// TwinCAT 3 PLC project Untitled1
// ProgramVersion: 3.1.4024.0
// libraries:
//   Tc2_Standard, * (Beckhoff Automation GmbH)
//   Tc2_System, * (Beckhoff Automation GmbH)
//   Tc3_Module, * (Beckhoff Automation GmbH)
// project tree:
//   / GlobalTextList.TcGTLO (not stored), PlcTask.TcTTO (not stored), Visualization Manager.TcVMO (not stored)
//   GVLs/ GIOL.TcGVL (not stored), Global_IO_assignment.TcPOU (not stored), GVL.TcGVL (not stored)
//   POUs/ MAIN.TcPOU, INMODE.TcPOU (not stored)
//   VISUs/ StandardPLCversenyVISU.TcVIS
// real-time tasks:
//   TASK PlcTask: cycle T#10ms, priority 20, ADS port 350
// I/O:
//   DEVICE Device 1 (EtherCAT), AmsNetId 5.86.98.224.2.1
//     Term 1 (EK1200) [EK1200-5000 EtherCAT Power supply (2A E-Bus)]
//       Term 2 (EL1008) [EL1008 8Ch. Dig. Input 24V, 3ms]
//       Term 3 (EL1008) [EL1008 8Ch. Dig. Input 24V, 3ms]
//       Term 4 (EL2008) [EL2008 8Ch. Dig. Output 24V, 0.5A]
//       Term 5 (EL2008) [EL2008 8Ch. Dig. Output 24V, 0.5A]
//       Term 6 (EL9011) [EL9011 End Terminal]
// variable links:
//   Untitled1/Untitled1 Instance <-> Device 1 (EtherCAT)/Term 1 (EK1200)/Term 2 (EL1008)
//     PlcTask Inputs/GIOL.xIn{0..7} <-> Channel {1..8}/Input  (8 links)
//   Untitled1/Untitled1 Instance <-> Device 1 (EtherCAT)/Term 1 (EK1200)/Term 3 (EL1008)
//     PlcTask Inputs/GIOL.xIn{8..15} <-> Channel {1..8}/Input  (8 links)
//   Untitled1/Untitled1 Instance <-> Device 1 (EtherCAT)/Term 1 (EK1200)/Term 4 (EL2008)
//     PlcTask Outputs/GIOL.Out{0..7} <-> Channel {1..8}/Output  (8 links)
//   Untitled1/Untitled1 Instance <-> Device 1 (EtherCAT)/Term 1 (EK1200)/Term 5 (EL2008)
//     PlcTask Outputs/GIOL.Out{8..15} <-> Channel {1..8}/Output  (8 links)

// ---- POUs/MAIN.TcPOU
PROGRAM MAIN
VAR
	INMODE : INMODE;
END_VAR

INMODE(); 
CASE GIOL.CaseNum OF
	0:GIOL.TaskName:="First Tsak";
	10:GIOL.TaskName:="Second Tsak";
	20:GIOL.TaskName:="Third Tsak";
	30:GIOL.TaskName:="Fourth Tsak";
	40:GIOL.TaskName:="Fifth Tsak";
	50:GIOL.TaskName:="Sixth Tsak";
	ELSE
		GIOL.CaseNum:=0;
END_CASE

END_PROGRAM

// ---- VISUs/StandardPLCversenyVISU.TcVIS
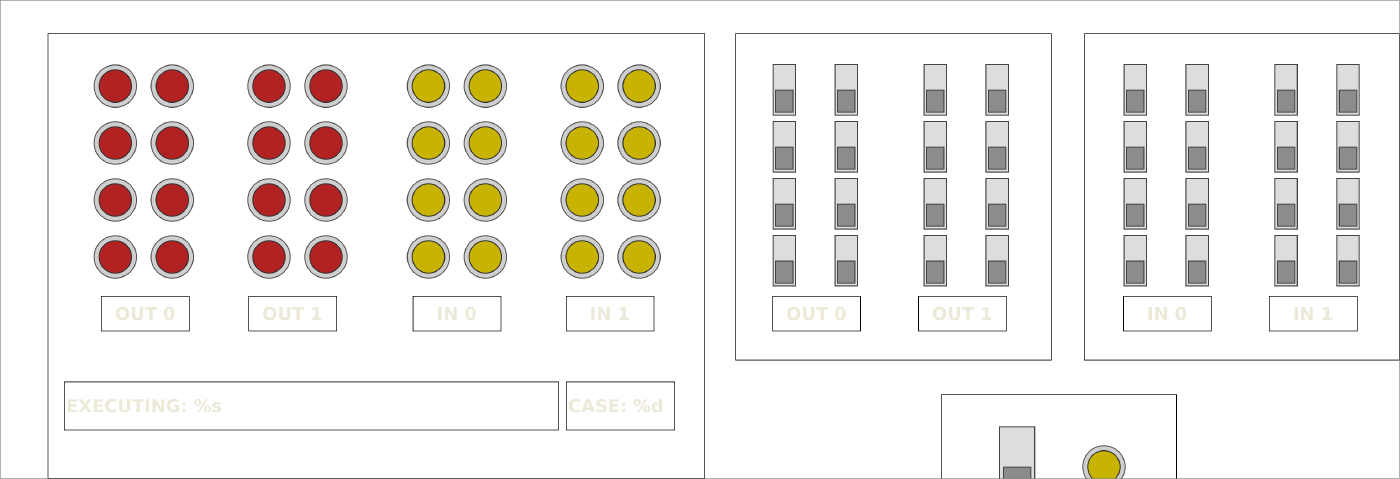
VISUALIZATION StandardPLCversenyVISU  // 1967x673
    Rectangle (1322,554 331x259)
    Rectangle (1033,47 444x459)
    Rectangle (67,47 923x626)
    Lamp1 (127,86 70x70), variable: GIOL.out0, style: Lamp-Lamp1-Red
    Lamp1 (207,86 70x70), variable: GIOL.out1, style: Lamp-Lamp1-Red
    Lamp1 (343,86 70x70), variable: GIOL.out8, style: Lamp-Lamp1-Red
    Lamp1 (423,86 70x70), variable: GIOL.out9, style: Lamp-Lamp1-Red
    Lamp1 (127,166 70x70), variable: GIOL.out2, style: Lamp-Lamp1-Red
    Lamp1 (207,166 70x70), variable: GIOL.out3, style: Lamp-Lamp1-Red
    Lamp1 (343,166 70x70), variable: GIOL.out10, style: Lamp-Lamp1-Red
    Lamp1 (423,166 70x70), variable: GIOL.out11, style: Lamp-Lamp1-Red
    Lamp1 (127,246 70x70), variable: GIOL.out4, style: Lamp-Lamp1-Red
    Lamp1 (207,246 70x70), variable: GIOL.out5, style: Lamp-Lamp1-Red
    Lamp1 (343,246 70x70), variable: GIOL.out12, style: Lamp-Lamp1-Red
    Lamp1 (423,246 70x70), variable: GIOL.out13, style: Lamp-Lamp1-Red
    Lamp1 (127,326 70x70), variable: GIOL.out6, style: Lamp-Lamp1-Red
    Lamp1 (207,326 70x70), variable: GIOL.out7, style: Lamp-Lamp1-Red
    Lamp1 (343,326 70x70), variable: GIOL.out14, style: Lamp-Lamp1-Red
    Lamp1 (423,326 70x70), variable: GIOL.out15, style: Lamp-Lamp1-Red
    Lamp1 (567,86 70x70), variable: GIOL.in0, style: Lamp-Lamp1-Yellow
    Lamp1 (647,86 70x70), variable: GIOL.in1, style: Lamp-Lamp1-Yellow
    Lamp1 (783,86 70x70), variable: GIOL.in8, style: Lamp-Lamp1-Yellow
    Lamp1 (863,86 70x70), variable: GIOL.in9, style: Lamp-Lamp1-Yellow
    Lamp1 (567,166 70x70), variable: GIOL.in2, style: Lamp-Lamp1-Yellow
    Lamp1 (647,166 70x70), variable: GIOL.in3, style: Lamp-Lamp1-Yellow
    Lamp1 (783,166 70x70), variable: GIOL.in10, style: Lamp-Lamp1-Yellow
    Lamp1 (863,166 70x70), variable: GIOL.in11, style: Lamp-Lamp1-Yellow
    Lamp1 (567,246 70x70), variable: GIOL.in4, style: Lamp-Lamp1-Yellow
    Lamp1 (647,246 70x70), variable: GIOL.in5, style: Lamp-Lamp1-Yellow
    Lamp1 (783,246 70x70), variable: GIOL.in12, style: Lamp-Lamp1-Yellow
    Lamp1 (863,246 70x70), variable: GIOL.in13, style: Lamp-Lamp1-Yellow
    Lamp1 (567,326 70x70), variable: GIOL.in6, style: Lamp-Lamp1-Yellow
    Lamp1 (647,326 70x70), variable: GIOL.in7, style: Lamp-Lamp1-Yellow
    Lamp1 (783,326 70x70), variable: GIOL.in14, style: Lamp-Lamp1-Yellow
    Lamp1 (863,326 70x70), variable: GIOL.in15, style: Lamp-Lamp1-Yellow
    Rectangle (349,416 124x49), "OUT 1"
    Rectangle (580,416 124x49), "IN 0"
    Rectangle (142,416 124x49), "OUT 0"
    Rectangle (795,416 124x49), "IN 1"
    Rectangle (90,536 695x68), "EXECUTING: %s", text variable: GIOL.TaskName
    DipSwitch (1153,86 72x80), variable: GIOL.out1, behaviour: TOGGLE, style: Switch-DipSwitch-Gray
    DipSwitch (1066,86 72x80), variable: GIOL.out0, behaviour: TOGGLE, style: Switch-DipSwitch-Gray
    DipSwitch (1153,166 72x80), variable: GIOL.out3, behaviour: TOGGLE, style: Switch-DipSwitch-Gray
    DipSwitch (1066,166 72x80), variable: GIOL.out2, behaviour: TOGGLE, style: Switch-DipSwitch-Gray
    DipSwitch (1153,246 72x80), variable: GIOL.out5, behaviour: TOGGLE, style: Switch-DipSwitch-Gray
    DipSwitch (1066,246 72x80), variable: GIOL.out4, behaviour: TOGGLE, style: Switch-DipSwitch-Gray
    DipSwitch (1153,326 72x80), variable: GIOL.out7, behaviour: TOGGLE, style: Switch-DipSwitch-Gray
    DipSwitch (1066,326 72x80), variable: GIOL.out6, behaviour: TOGGLE, style: Switch-DipSwitch-Gray
    DipSwitch (1365,86 72x80), variable: GIOL.out9, behaviour: TOGGLE, style: Switch-DipSwitch-Gray
    DipSwitch (1278,86 72x80), variable: GIOL.out8, behaviour: TOGGLE, style: Switch-DipSwitch-Gray
    DipSwitch (1365,166 72x80), variable: GIOL.out11, behaviour: TOGGLE, style: Switch-DipSwitch-Gray
    DipSwitch (1278,166 72x80), variable: GIOL.out10, behaviour: TOGGLE, style: Switch-DipSwitch-Gray
    DipSwitch (1365,246 72x80), variable: GIOL.out13, behaviour: TOGGLE, style: Switch-DipSwitch-Gray
    DipSwitch (1278,246 72x80), variable: GIOL.out12, behaviour: TOGGLE, style: Switch-DipSwitch-Gray
    DipSwitch (1365,326 72x80), variable: GIOL.out15, behaviour: TOGGLE, style: Switch-DipSwitch-Gray
    DipSwitch (1278,326 72x80), variable: GIOL.out14, behaviour: TOGGLE, style: Switch-DipSwitch-Gray
    Rectangle (1290,416 124x49), "OUT 1"
    Rectangle (1085,416 124x49), "OUT 0"
    Rectangle (1523,47 444x459)
    DipSwitch (1646,86 72x80), variable: GIOL.bIn1, behaviour: TOGGLE, style: Switch-DipSwitch-Gray
    DipSwitch (1559,86 72x80), variable: GIOL.bIn0, behaviour: TOGGLE, style: Switch-DipSwitch-Gray
    DipSwitch (1646,166 72x80), variable: GIOL.bIn3, behaviour: TOGGLE, style: Switch-DipSwitch-Gray
    DipSwitch (1559,166 72x80), variable: GIOL.bIn2, behaviour: TOGGLE, style: Switch-DipSwitch-Gray
    DipSwitch (1646,246 72x80), variable: GIOL.bIn5, behaviour: TOGGLE, style: Switch-DipSwitch-Gray
    DipSwitch (1559,246 72x80), variable: GIOL.bIn4, behaviour: TOGGLE, style: Switch-DipSwitch-Gray
    DipSwitch (1646,326 72x80), variable: GIOL.bIn7, behaviour: TOGGLE, style: Switch-DipSwitch-Gray
    DipSwitch (1559,326 72x80), variable: GIOL.bIn6, behaviour: TOGGLE, style: Switch-DipSwitch-Gray
    DipSwitch (1858,86 72x80), variable: GIOL.bIn9, behaviour: TOGGLE, style: Switch-DipSwitch-Gray
    DipSwitch (1771,86 72x80), variable: GIOL.bIn8, behaviour: TOGGLE, style: Switch-DipSwitch-Gray
    DipSwitch (1858,166 72x80), variable: GIOL.bIn11, behaviour: TOGGLE, style: Switch-DipSwitch-Gray
    DipSwitch (1771,166 72x80), variable: GIOL.bIn10, behaviour: TOGGLE, style: Switch-DipSwitch-Gray
    DipSwitch (1858,246 72x80), variable: GIOL.bIn13, behaviour: TOGGLE, style: Switch-DipSwitch-Gray
    DipSwitch (1771,246 72x80), variable: GIOL.bIn12, behaviour: TOGGLE, style: Switch-DipSwitch-Gray
    DipSwitch (1858,326 72x80), variable: GIOL.bIn15, behaviour: TOGGLE, style: Switch-DipSwitch-Gray
    DipSwitch (1771,326 72x80), variable: GIOL.bIn14, behaviour: TOGGLE, style: Switch-DipSwitch-Gray
    Rectangle (1783,416 124x49), "IN 1"
    Rectangle (1578,416 124x49), "IN 0"
    Rectangle (795,536 153x68), "CASE: %d", text variable: GIOL.CaseNum
    DipSwitch (1371,599 116x113), variable: MAIN.INMODE.INState, behaviour: TOGGLE, style: Switch-DipSwitch-Gray
    Rectangle (1381,744 226x49), "INPUT MODE"
    Lamp1 (1516,621 70x70), variable: MAIN.INMODE.INState, style: Lamp-Lamp1-Yellow
END_VISUALIZATION
